TYPE SRecoveryRequestOutput EXTENDS STriggeredOutput :
STRUCT
	RequestedState: STRING(256);
END_STRUCT
END_TYPE

(* stored: Version 1.1.0.1, ProductVersion 3.1.4024.9
   DUT SRecoveryRequestOutput: Id {ec4553f3-e045-4212-85e5-e2ee6ad8c437} *)
